FUNCTION_BLOCK HydraulicsPumpsGroupIO EXTENDS SM_HydraulicsPumpsGroupIO
VAR_INPUT
END_VAR
VAR_OUTPUT
END_VAR
VAR
END_VAR

SUPER^();

END_FUNCTION_BLOCK

(* stored: Version 1.1.0.1, ProductVersion 3.1.4018.5
   POU HydraulicsPumpsGroupIO: Id {bad74441-994e-487f-abea-96b273d9c376}, SpecialFunc None *)
